{attribute 'pack_mode' := '2'}
TYPE ST_GEAR_DATA :
STRUCT
  rDeltaToMasterPos       : REAL;
  rModuloSyncPosSlave     : REAL;
  rMasterStartDistance    : REAL;
  rGearNumerator          : REAL;
  iGearDenumerator        : USINT  := 1;
END_STRUCT
END_TYPE

(* stored: Version 1.1.0.1, ProductVersion 3.1.4024.15
   DUT ST_GEAR_DATA: Id {058e7510-a7ec-4bcf-bb55-c337667a6f5b} *)
